{attribute 'linkalways'} 
{attribute 'no_explicit_call' := 'This FB is a CLASS and must be accessed using methods or properties'}
{attribute 'enable_dynamic_creation'}
FUNCTION_BLOCK _TIME_OF_DAY EXTENDS DatatypeBase
VAR
	localData : TIME_OF_DAY;
	activeData : REFERENCE TO TIME_OF_DAY REF= localData;
END_VAR

PROPERTY PUBLIC Address : PVOID
GET
Address := ADR(activeData);
END_GET
END_PROPERTY

METHOD PUBLIC ClearReference
VAR_INPUT
END_VAR
activeData REF= localData;
END_METHOD

METHOD PUBLIC Clone : I_Datatype
VAR
    pClone : POINTER TO _TIME_OF_DAY;
END_VAR
pClone := __NEW(_TIME_OF_DAY(InitialValue := Value));
Clone := pClone^;
END_METHOD

METHOD FB_init : BOOL
VAR_INPUT
	bInitRetains : BOOL; // if TRUE, the retain variables are initialized (warm start / cold start)
	bInCopyCode : BOOL;  // if TRUE, the instance afterwards gets moved WORDo the copy code (online change)
	InitialValue : TIME_OF_DAY;
END_VAR
localData := InitialValue;
END_METHOD

METHOD PUBLIC MakeReferenceTo
VAR_INPUT
	ReferenceTarget : REFERENCE TO TIME_OF_DAY;
END_VAR
activeData REF= ReferenceTarget;
END_METHOD

METHOD PUBLIC SerializeWith
VAR_INPUT
	Serializer : I_Serializer;
END_VAR
Serializer.AddTod(activeData);
END_METHOD

PROPERTY PUBLIC Size : UDINT
GET
Size := SIZEOF(activeData);
END_GET
END_PROPERTY

METHOD TryDeserializeFrom : BOOL
VAR_INPUT
	Deserializer : I_Deserializer;
	Feedback : I_DeserializerFeedback;
END_VAR
TryDeserializeFrom := Deserializer.TryGetTod(activeData, Feedback);
END_METHOD

METHOD TryMakeReferenceTo : BOOL
VAR_INPUT
	Target : I_Datatype;
END_VAR
VAR
	pTargetData : POINTER TO TIME_OF_DAY;
END_VAR
IF NOT (Target.TypeName = TypeName) THEN
	RETURN;
END_IF

pTargetData := Target.Address;
activeData REF= pTargetData^;
TryMakeReferenceTo := TRUE;
END_METHOD

PROPERTY PUBLIC TypeName : T_MAXSTRING
GET
TypeName := 'TIME_OF_DAY';
END_GET
END_PROPERTY

PROPERTY PUBLIC Value : REFERENCE TO TIME_OF_DAY
GET
Value REF= activeData;
END_GET
END_PROPERTY

END_FUNCTION_BLOCK

(* stored: Version 1.1.0.1, ProductVersion 3.1.4024.13
   POU _TIME_OF_DAY: Id {4b0a87e2-c072-49e3-85b6-cf5a09ecca1b}, SpecialFunc None
   Folder Constructor: Id {fe765294-52a3-4cc6-9810-ab5fce0b0b56}
   Property Address: Id {d5191e00-79ef-4b73-93f9-3dad019fc62c}
   Get Get: Id {01b1b2c4-06eb-4dba-865f-63a3bd9811a8}
   Method ClearReference: Id {a52a591c-35c8-46b5-bdc1-372072302e7d}
   Method Clone: Id {ca8a7919-55f6-4ff5-9430-f60c7898a25c}
   Method FB_init: Id {1fbdcfce-b279-473b-9b76-6271e98891a6}
   Method MakeReferenceTo: Id {8c3e3545-8418-445f-b0b5-e63df29f9f12}
   Method SerializeWith: Id {3241cf62-0bc9-4f29-8528-4ca6afca0c33}
   Property Size: Id {7c1cac0a-59aa-44d1-af3e-9643522a3ad5}
   Get Get: Id {bea81c82-5c49-4ce2-a35d-4fee953004a3}
   Method TryDeserializeFrom: Id {e842ce0e-8e12-488b-a930-d97ef3d9e171}
   Method TryMakeReferenceTo: Id {2779fd4c-0763-41ec-958d-b150f3e80d4d}
   Property TypeName: Id {9d8a6a96-27e0-47a7-ab38-5d7fea91fb21}
   Get Get: Id {b55c9afd-0777-4ab9-aa4c-1eb76ae24a11}
   Property Value: Id {22db774c-0d72-46b4-a6e3-91de72a2a61b}
   Get Get: Id {2e0726c9-a86a-40aa-95b6-50838455feba} *)
